# EPICS substitutions: db/Beckhoff_1XXX/ecmcEP1918-0002_ALVIN_OBSOLETE.substitutions
file "ecmc_binaryOutput-chX.template" { pattern
  { CH_ID }
  { 1     }
  { 2     }
  { 3     }
  { 4     }
  { 5     }
  { 6     }
  { 7     }
  { 8     }
}

file "ecmc_controlWord-chX.template" { pattern
  { CH_ID }
  { 1     }
  { 2     }
  { 3     }
  { 4     }
  { 5     }
  { 6     }
  { 7     }
}

file "ecmc_status-chX.template" { pattern
  { CH_ID, KEY }
  { 1,     ""  }
  { 2,     ""  }
  { 3,     ""  }
  { 4,     ""  }
  { 5,     ""  }
}
